FUNCTION_BLOCK FILTER_JSON_TIMESERIES
  {SET_ATTRIBUTE(OpcUa, POINT.ENDPOINT)}
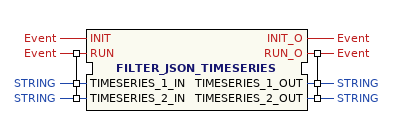
  EVENT_INPUT
    INIT;
    RUN WITH TIMESERIES_1_IN, TIMESERIES_2_IN;
  END_EVENT
  EVENT_OUTPUT
    INIT_O;
    RUN_O WITH TIMESERIES_1_OUT, TIMESERIES_2_OUT;
  END_EVENT
  VAR_INPUT
    TIMESERIES_1_IN : STRING; {SET_ATTRIBUTE(OpcUa, Variable)}
    TIMESERIES_2_IN : STRING; {SET_ATTRIBUTE(OpcUa, Variable)}
  END_VAR
  VAR_OUTPUT
    TIMESERIES_1_OUT : STRING; {SET_ATTRIBUTE(OpcUa, Variable)}
    TIMESERIES_2_OUT : STRING; {SET_ATTRIBUTE(OpcUa, Variable)}
  END_VAR
END_FUNCTION_BLOCK
